{attribute addProperty BoxType "AX8206-0000-0041-0041"}
{attribute addProperty Id "DeviceDevice_FD48B4B01620Ch_ACh_A_99F8614F240300Ch_BCh_B_5DC205AF240300WcStateAT %I*WcState_F855686C1620InfoDataAT %I*InfoData_17277C5A208260"}
{attribute addProperty CRC "451800211"}
{attribute addProperty SizeInBites "720"}
{attribute addProperty SizeInBytes "90"}
TYPE AX8206_D62D6325 :
STRUCT
	{attribute addProperty Name "Device"}
	Device : Device_FD48B4B0;
	{attribute addProperty Name "Ch_A"}
	Ch_A : Ch_A_99F8614F;
	{attribute addProperty Name "Ch_B"}
	Ch_B : Ch_B_5DC205AF;
	{attribute addProperty Name "WcState"}
	WcState : WcState_F855686C;
	{attribute addProperty Name "InfoData"}
	InfoData : InfoData_17277C5A;
END_STRUCT
END_TYPE

(* stored: Version 1.2.0.0, ProductVersion 3.1.4024.9
   DUT AX8206_D62D6325: Id {8b4aecd0-a8af-450c-8d97-f0d3fdd731f5} *)
